Fanuc KAREL source: CNV_CNF_STRG.kl

PROGRAM T
%NOLOCKGROUP
VAR
 v0 : CONFIG
 v1 : STRING[40]
 v2 : INTEGER
 v3 : INTEGER
BEGIN
 CNV_CNF_STRG(v0, v1, v2, v3)
END T
